// Mitsubishi GX Works2 project: LRI - Sinal de Pulso   PLC: Q03UDV
// HelloWorld

PROGRAM MAIN
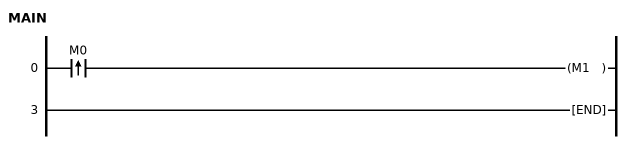
0     LDP     M0
      OUT     M1
3     END
END_PROGRAM
